PROGRAM valve_digital_control
VAR PERSISTENT
	// Example digital valve
	nv_3372: valve_digital;
END_VAR

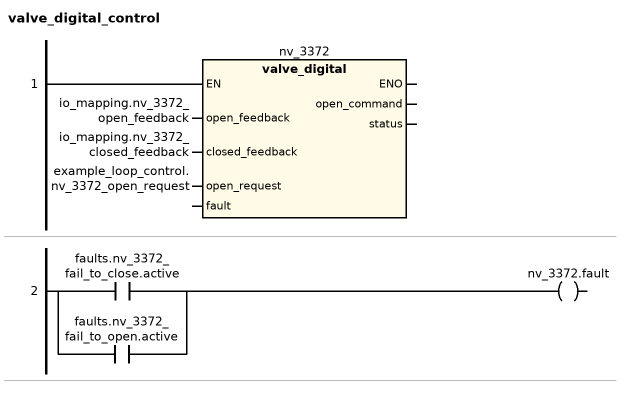
// NETWORK 1
nv_3372(
    open_feedback := io_mapping.nv_3372_open_feedback,
    closed_feedback := io_mapping.nv_3372_closed_feedback,
    open_request := example_loop_control.nv_3372_open_request); // valve_digital

// NETWORK 2
nv_3372.fault := faults.nv_3372_fail_to_close.active OR faults.nv_3372_fail_to_open.active;

END_PROGRAM

(* stored: Version 1.1.0.1, ProductVersion 3.1.4024.12
   POU valve_digital_control: Id {877f0e18-5c71-495f-9644-351f8ecc5f44}, SpecialFunc None *)
